{attribute 'qualified_only'}
VAR_GLOBAL
	
	q_relaisTest : BOOL;
	
	i_fotoCel : BOOL;
	
END_VAR

(* stored: Version 1.1.0.1, ProductVersion 3.1.4024.12
   GVL Alias: Id {125f7c14-bc07-4185-8080-6bf9d7d4c446} *)
